(* LS Electric XG5000 project: 커피창린스PLC *)
(* PLC LSPLC *)

PROGRAM NewProgram (* task: 스캔 프로그램 *)
VAR
    T1 : TON;
    T2 : TON;
    근접센서1 AT %MX7 : BOOL;
    근접센서2 : BOOL;
    대형1층동작 : TON;
    대형감지 AT %MX2 : BOOL;
    대형감지완료 AT %MX5 : BOOL;
    대형도착 AT %QX0.1.8 : BOOL;
    대형엘리도착 : BOOL;
    대형엘리동작1 : TON;
    대형입장 AT %IX0.0.2 : BOOL;
    도착 AT %QX0.1.13 : BOOL;
    레일동작 AT %QX0.1.4 : BOOL;
    레일정지 AT %QX0.1.5 : BOOL;
    소형감지 AT %MX0 : BOOL;
    소형감지완료 AT %MX3 : BOOL;
    소형도착 AT %QX0.1.6 : BOOL;
    소형입장 AT %IX0.0.0 : BOOL;
    실링기계 : TON;
    실링기계동작 : BOOL;
    실링레일 : TON;
    실링레일동작 : BOOL;
    엘리1층도착 : BOOL;
    엘리내려감 AT %QX0.1.11 : BOOL;
    엘리베이터대기 : TON;
    엘리베이터동작 AT %QX0.1.9 : BOOL;
    엘리베이터중지 AT %QX0.1.10 : BOOL;
    자동차입장감지센서 AT %QX0.1.0 : BOOL;
    자동차퇴장감지 AT %IX0.0.4 : BOOL;
    자동차퇴장알림 AT %QX0.1.12 : BOOL;
    주차차단기개방 AT %QX0.1.1 : BOOL;
    주차차단기차단 : BOOL;
    중형1층동작 : TON;
    중형감지 AT %MX1 : BOOL;
    중형감지완료 AT %MX4 : BOOL;
    중형도착 AT %QX0.1.7 : BOOL;
    중형엘리도착 : BOOL;
    중형엘리동작1 : TON;
    중형입장 AT %IX0.0.1 : BOOL;
    지나감감지 : TON;
    커피배달중 AT %QX0.1.14 : BOOL;
    커피제작시작 AT %QX0.1.2 : BOOL;
    커피제작완료 AT %QX0.1.3 : BOOL;
    커피주문 AT %IX0.0.3 : BOOL;
    커피주문완료 AT %MX6 : BOOL;
    퇴장알림 : TON;
END_VAR
VAR
    _p1 : BOOL;
END_VAR

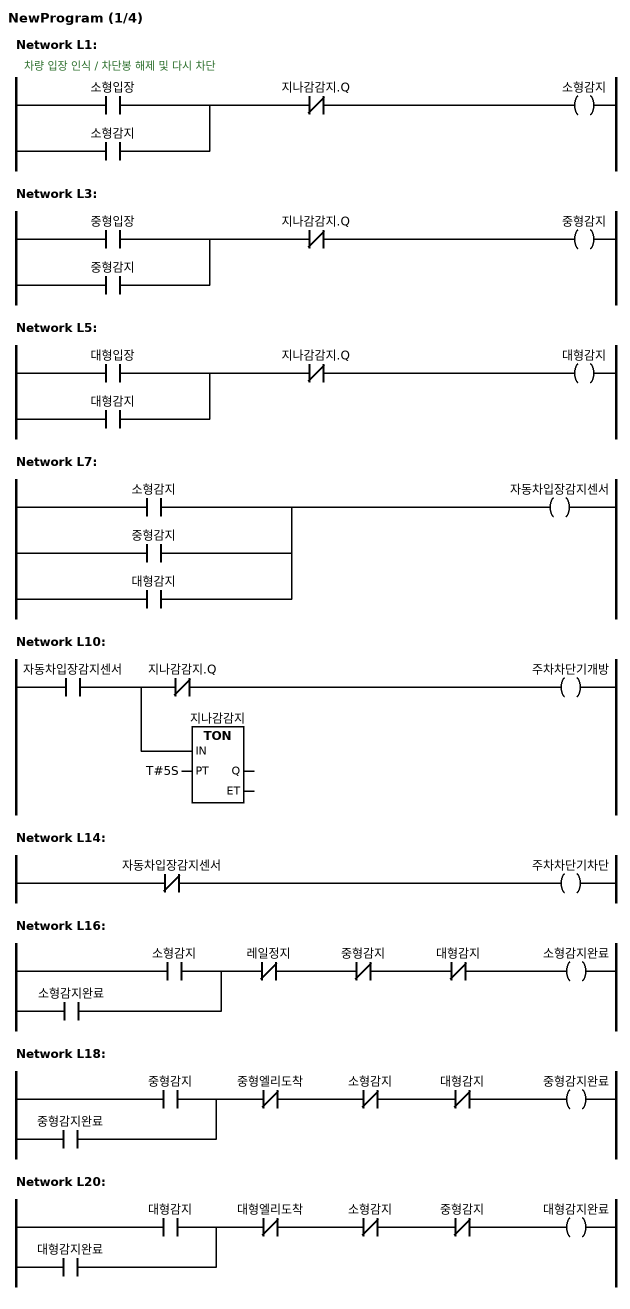
(* 차량 입장 인식 / 차단봉 해제 및 다시 차단 *)
(* Rung L1 *)
소형감지 := (소형입장 OR 소형감지) AND NOT 지나감감지.Q;
(* Rung L3 *)
중형감지 := (중형입장 OR 중형감지) AND NOT 지나감감지.Q;
(* Rung L5 *)
대형감지 := (대형입장 OR 대형감지) AND NOT 지나감감지.Q;
(* Rung L7 *)
자동차입장감지센서 := 소형감지 OR 중형감지 OR 대형감지;
(* Rung L10 *)
주차차단기개방 := 자동차입장감지센서 AND NOT 지나감감지.Q;
지나감감지(IN := 자동차입장감지센서, PT := T#5S);
(* Rung L14 *)
주차차단기차단 := NOT 자동차입장감지센서;
(* Rung L16 *)
소형감지완료 := (소형감지 OR 소형감지완료) AND NOT 레일정지 AND NOT 중형감지 AND NOT 대형감지;
(* Rung L18 *)
중형감지완료 := (중형감지 OR 중형감지완료) AND NOT 중형엘리도착 AND NOT 소형감지 AND NOT 대형감지;
(* Rung L20 *)
대형감지완료 := (대형감지 OR 대형감지완료) AND NOT 대형엘리도착 AND NOT 소형감지 AND NOT 중형감지;

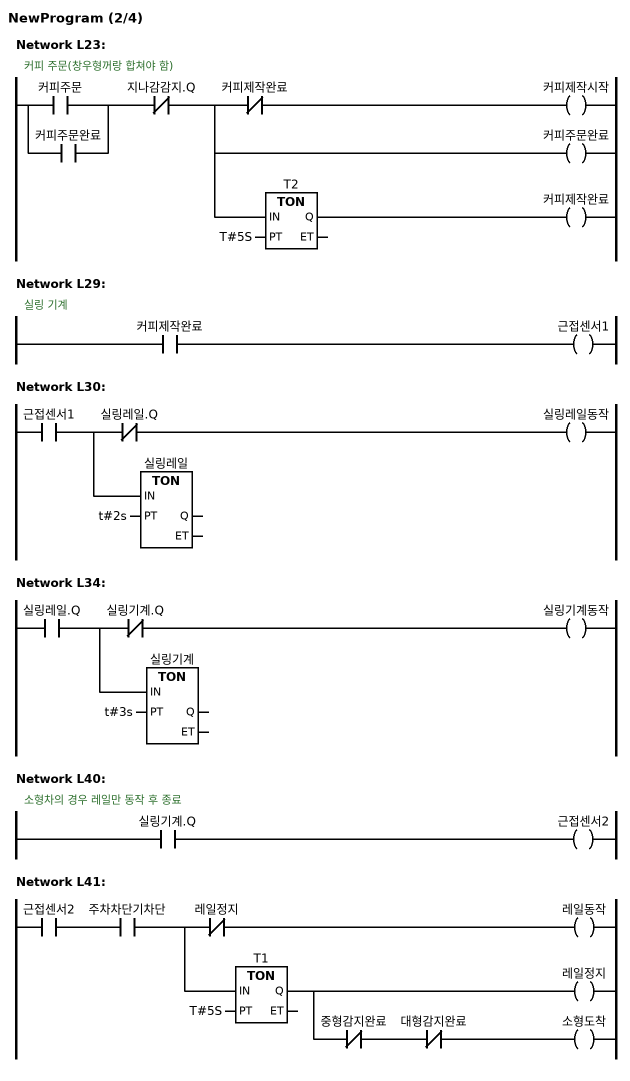
(* 커피 주문(창우형꺼랑 합쳐야 함) *)
(* Rung L23 *)
커피제작시작 := (커피주문 OR 커피주문완료) AND NOT 지나감감지.Q AND NOT 커피제작완료;
_p1 := (커피주문 OR 커피주문완료) AND NOT 지나감감지.Q;
커피주문완료 := _p1;
T2(IN := _p1, PT := T#5S);
커피제작완료 := T2.Q;
(* 실링 기계 *)
(* Rung L29 *)
근접센서1 := 커피제작완료;
(* Rung L30 *)
실링레일동작 := 근접센서1 AND NOT 실링레일.Q;
실링레일(IN := 근접센서1, PT := t#2s);
(* Rung L34 *)
실링기계동작 := 실링레일.Q AND NOT 실링기계.Q;
실링기계(IN := 실링레일.Q, PT := t#3s);
(* 소형차의 경우 레일만 동작 후 종료 *)
(* Rung L40 *)
근접센서2 := 실링기계.Q;
(* Rung L41 *)
레일동작 := 근접센서2 AND 주차차단기차단 AND NOT 레일정지;
T1(IN := 근접센서2 AND 주차차단기차단, PT := T#5S);
레일정지 := T1.Q;
소형도착 := T1.Q AND NOT 중형감지완료 AND NOT 대형감지완료;

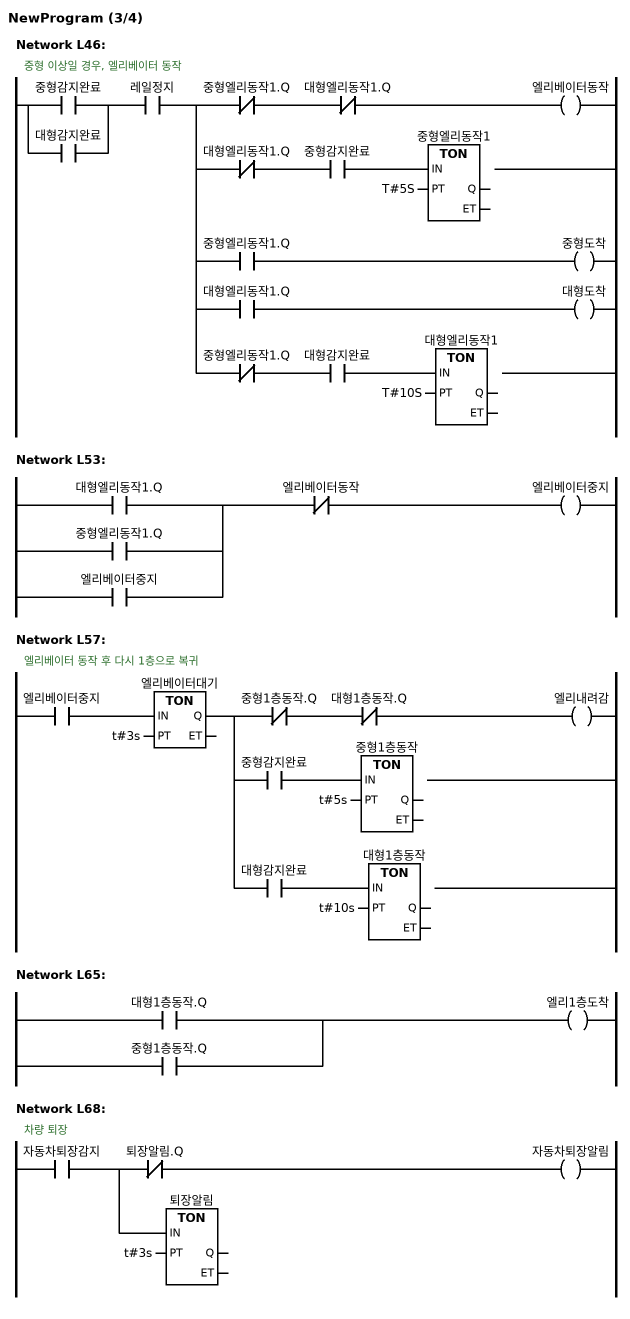
(* 중형 이상일 경우, 엘리베이터 동작 *)
(* Rung L46 *)
엘리베이터동작 := (중형감지완료 OR 대형감지완료) AND 레일정지 AND NOT 중형엘리동작1.Q AND NOT 대형엘리동작1.Q;
중형엘리동작1(IN := (중형감지완료 OR 대형감지완료) AND 레일정지 AND NOT 대형엘리동작1.Q AND 중형감지완료, PT := T#5S);
중형도착 := (중형감지완료 OR 대형감지완료) AND 레일정지 AND 중형엘리동작1.Q;
대형도착 := (중형감지완료 OR 대형감지완료) AND 레일정지 AND 대형엘리동작1.Q;
대형엘리동작1(IN := (중형감지완료 OR 대형감지완료) AND 레일정지 AND NOT 중형엘리동작1.Q AND 대형감지완료, PT := T#10S);
(* Rung L53 *)
엘리베이터중지 := (대형엘리동작1.Q OR 중형엘리동작1.Q OR 엘리베이터중지) AND NOT 엘리베이터동작;
(* 엘리베이터 동작 후 다시 1층으로 복귀 *)
(* Rung L57 *)
엘리베이터대기(IN := 엘리베이터중지, PT := t#3s);
엘리내려감 := 엘리베이터대기.Q AND NOT 중형1층동작.Q AND NOT 대형1층동작.Q;
중형1층동작(IN := 엘리베이터대기.Q AND 중형감지완료, PT := t#5s);
대형1층동작(IN := 엘리베이터대기.Q AND 대형감지완료, PT := t#10s);
(* Rung L65 *)
엘리1층도착 := 대형1층동작.Q OR 중형1층동작.Q;
(* 차량 퇴장 *)
(* Rung L68 *)
자동차퇴장알림 := 자동차퇴장감지 AND NOT 퇴장알림.Q;
퇴장알림(IN := 자동차퇴장감지, PT := t#3s);

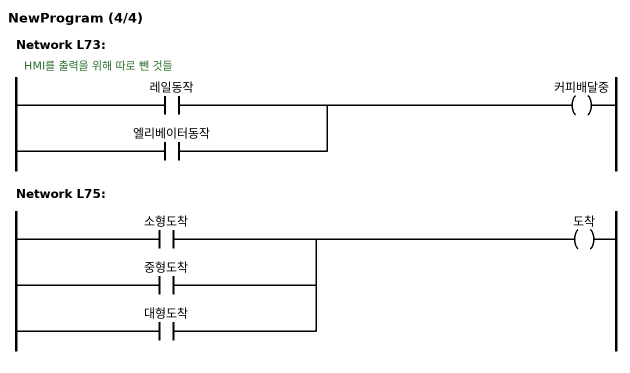
(* HMI를 출력을 위해 따로 뺀 것들 *)
(* Rung L73 *)
커피배달중 := 레일동작 OR 엘리베이터동작;
(* Rung L75 *)
도착 := 소형도착 OR 중형도착 OR 대형도착;
END_PROGRAM